Universal Robots PolyScope program: Impilacubi.urp

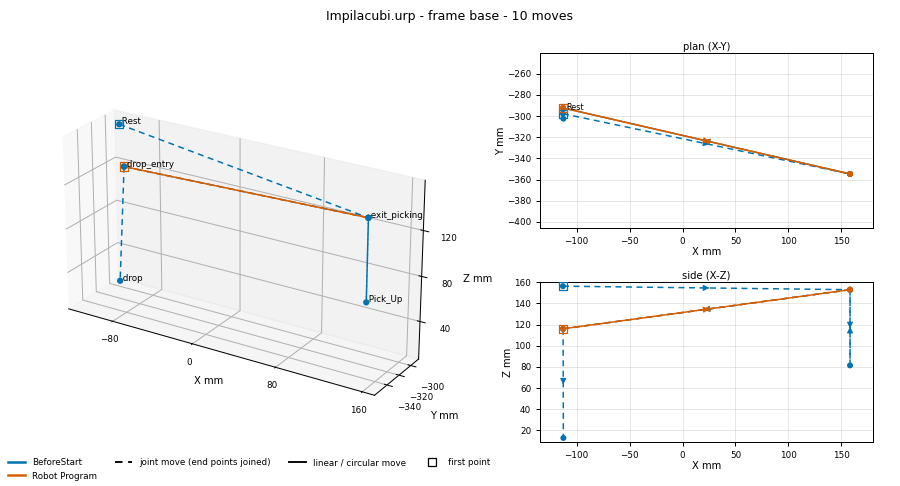
[picture p0: tool path of Impilacubi.urp in frame base, 10 of 12 moves have a stored position in this frame; points joined in program order, loops and branches not executed]
Program Impilacubi (installation=default directory=/programs createdIn=3.15.8.106339 lastSavedIn=3.15.8.106339 robotSerialNumber=2021330429)
Calibrated DH parameters: a=[-0.000156, -0.236402, -0.171625, 0.000006, -0.000047, 0]; d=[0.151683, 29.702709, 78.973085, -108.563557, 0.085229, 0.082167]; alpha=[1.57015, 0.001987, 0.001164, 1.571718, -1.571778, 0]; deltaTheta=[-0.000066, 0.24449, 0.39032, -0.635025, 0.000068, -0.000043]
BeforeStart
  URCap Gripper Activate (Robotiq_Grippers, Robotiq Inc.) dataModel(ResetAndActivateKey=false)
  URCap Gripper (Robotiq_Grippers, Robotiq Inc.) dataModel(position=0.0, force=0.0, speed=100.0, positionInDouble=0.0, forceInDouble=0.0, speedInDouble=100.0, slaveIds=[9], blocking=true)
  MoveJ speed 60 deg/s, acceleration 80 deg/s^2 (useActiveTCP=true)
    Waypoint Rest: TCP in base x=-112.987 y=-297.7 z=156.26 mm, rx=-2.2222 ry=-2.2185 rz=-0.0001 rad; joints [-90, -89.999, -89.999, -89.998, 90, 89.996] deg; flange x=-112.824 y=-297.877 z=313.26 mm, rx=-2.2222 ry=-2.2185 rz=-0.0001 rad
  MoveJ speed 60 deg/s, acceleration 80 deg/s^2 (useActiveTCP=true)
    Waypoint exit_picking: TCP in base x=158.29 y=-354.64 z=152.934 mm, rx=-0.0138 ry=3.0963 rz=-0.0574 rad; joints [-49.441, -104.465, -75.807, -86.383, 90.676, 39.971] deg; flange x=151.249 y=-348.853 z=309.67 mm, rx=-0.0138 ry=3.0963 rz=-0.0574 rad
  MoveJ speed 60 deg/s, acceleration 80 deg/s^2 (useActiveTCP=true)
    Waypoint Pick_Up: TCP in base x=158.293 y=-354.629 z=81.389 mm, rx=-0.0136 ry=3.0962 rz=-0.0575 rad; joints [-49.442, -107.285, -91.691, -67.674, 90.694, 39.996] deg; flange x=151.233 y=-348.838 z=238.124 mm, rx=-0.0136 ry=3.0962 rz=-0.0575 rad
  MoveJ speed 60 deg/s, acceleration 80 deg/s^2 (useActiveTCP=true)
    Waypoint exit_picking: TCP in base x=158.29 y=-354.64 z=152.934 mm, rx=-0.0138 ry=3.0963 rz=-0.0574 rad; joints [-49.441, -104.465, -75.807, -86.383, 90.676, 39.971] deg; flange x=151.249 y=-348.853 z=309.67 mm, rx=-0.0138 ry=3.0963 rz=-0.0574 rad
  MoveJ speed 60 deg/s, acceleration 80 deg/s^2 (useActiveTCP=true)
    Waypoint drop_entry: TCP in base x=-112.858 y=-292.299 z=116.007 mm, rx=2.2208 ry=2.2188 rz=-0.0063 rad; joints [-89.97, -89.32, -101.691, -78.665, 89.995, 89.996] deg; flange x=-112.665 y=-291.6 z=273.005 mm, rx=2.2208 ry=2.2188 rz=-0.0063 rad
  MoveJ speed 60 deg/s, acceleration 80 deg/s^2 (useActiveTCP=true)
    Waypoint drop: TCP in base x=-112.615 y=-302.416 z=12.836 mm, rx=2.2198 ry=2.2202 rz=-0.0065 rad; joints [-89.918, -102.763, -117.558, -49.36, 90.009, 90.015] deg; flange x=-112.374 y=-301.732 z=169.835 mm, rx=2.2198 ry=2.2202 rz=-0.0065 rad
  URCap Gripper Activate (Robotiq_Grippers, Robotiq Inc.) dataModel(ResetAndActivateKey=false)
  P := Pick_Up
  D := drop
  distance := 0.024
  Popup Message (haltProgram=false message=fine prestart inputType=Text)
Robot Program (runOnlyOnce=false)
  Loop Counting (count=4) loopVariable(name=Loop_2)
    MoveJ speed 60 deg/s, acceleration 80 deg/s^2 (useActiveTCP=true)
      Waypoint drop_entry: TCP in base x=-112.858 y=-292.299 z=116.007 mm, rx=2.2208 ry=2.2188 rz=-0.0063 rad; joints [-89.97, -89.32, -101.691, -78.665, 89.995, 89.996] deg; flange x=-112.665 y=-291.6 z=273.005 mm, rx=2.2208 ry=2.2188 rz=-0.0063 rad
    MoveJ speed 60 deg/s, acceleration 80 deg/s^2 (useActiveTCP=true)
      Waypoint exit_picking: TCP in base x=158.29 y=-354.64 z=152.934 mm, rx=-0.0138 ry=3.0963 rz=-0.0574 rad; joints [-49.441, -104.465, -75.807, -86.383, 90.676, 39.971] deg; flange x=151.249 y=-348.853 z=309.67 mm, rx=-0.0138 ry=3.0963 rz=-0.0574 rad
    MoveL speed 250 mm/s, acceleration 1200 mm/s^2 (useActiveTCP=true) feature=Base
      Waypoint Waypoint (Variable): variable=P
      URCap Gripper (Robotiq_Grippers, Robotiq Inc.) dataModel(position=100.0, force=0.0, speed=0.0, positionInDouble=100.0, forceInDouble=0.0, speedInDouble=0.0, slaveIds=[9], blocking=true)
    MoveL speed 250 mm/s, acceleration 1200 mm/s^2 (useActiveTCP=true) feature=Base
      Waypoint exit_picking: TCP in base x=158.29 y=-354.64 z=152.934 mm, rx=-0.0138 ry=3.0963 rz=-0.0574 rad; joints [-49.441, -104.465, -75.807, -86.383, 90.676, 39.971] deg; flange x=151.249 y=-348.853 z=309.67 mm, rx=-0.0138 ry=3.0963 rz=-0.0574 rad
    MoveL speed 250 mm/s, acceleration 1200 mm/s^2 (useActiveTCP=true) feature=Base
      Waypoint drop_entry: TCP in base x=-112.858 y=-292.299 z=116.007 mm, rx=2.2208 ry=2.2188 rz=-0.0063 rad; joints [-89.97, -89.32, -101.691, -78.665, 89.995, 89.996] deg; flange x=-112.665 y=-291.6 z=273.005 mm, rx=2.2208 ry=2.2188 rz=-0.0063 rad
    MoveL speed 250 mm/s, acceleration 1200 mm/s^2 (useActiveTCP=true) feature=Base
      Waypoint Waypoint (Variable): variable=D
      URCap Gripper (Robotiq_Grippers, Robotiq Inc.) dataModel(position=0.0, force=0.0, speed=0.0, positionInDouble=0.0, forceInDouble=0.0, speedInDouble=0.0, slaveIds=[9], blocking=true)
    Script: P[2]=P[2]-distance
    Script: D[2]=D[2]+(distance+0.005)
  If Loop_2≟4 (checkContinuously=true)
    D := drop
    P := Pick_Up
    Popup Message (haltProgram=false message=Fine impilamento inputType=Text)
